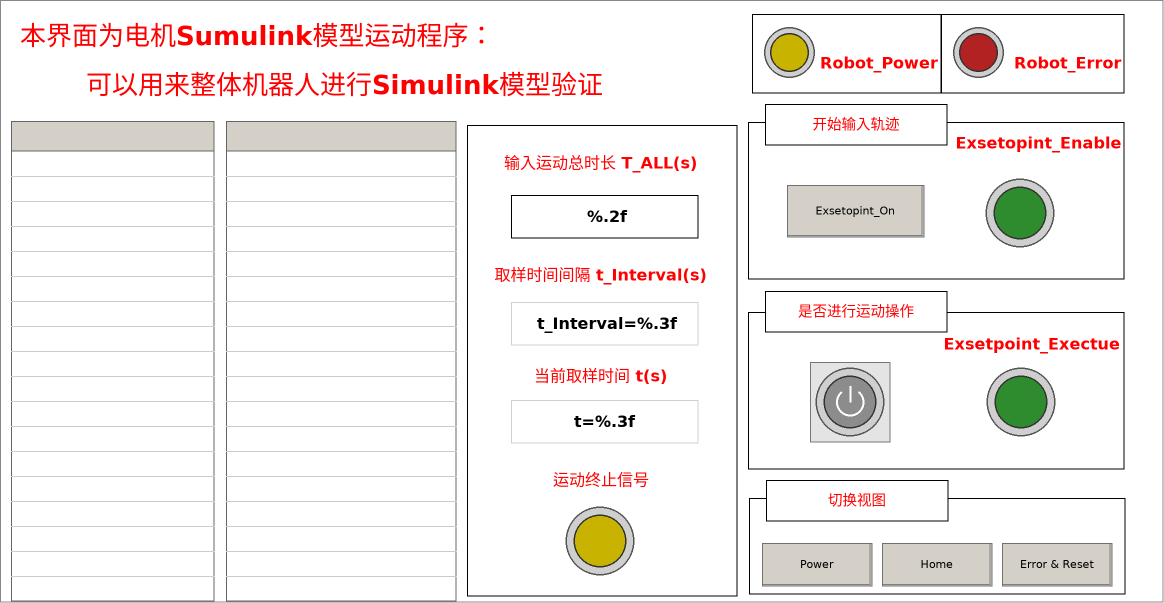
VISUALIZATION Visu_SimulinkMove  // 1164x603
    Rectangle (749,498 376x96)
    Rectangle (766,480 182x41), "切换视图"
    Button (762,543 110x43), "Power"
        OnMouseClick: change screen: Visu_Power
    Button (1002,543 110x43), "Error & Reset"
        OnMouseClick: change screen: Visu_Reset
    Button (882,543 110x43), "Home"
        OnMouseClick: change screen: Visu_Home
    Rectangle (467,125 270x471)
    Rectangle (752,14 189x79)
    Rectangle (748,312 376x157)
    Label (902,328 260x32), "Exsetpoint_Exectue"
    Rectangle (765,291 182x41), "是否进行运动操作"
    Lamp1 (981,362 80x80), variable: ExSetPoint_Execute, style: Lamp-Lamp1-Green
    PowerSwitch (810,362 80x80), variable: ExSetPoint_Execute, behaviour: TOGGLE, style: Switch-PowerSwitch-Gray
    Rectangle (941,14 183x79)
    Lamp1 (948,23 61x59), variable: Hexapod_Robot.Robot_Error, style: Lamp-Lamp1-Red
    Label (991,47 154x32), "Robot_Error"
    Label (17,15 572x42), "本界面为电机Sumulink模型运动程序："
    Label (83,64 874x42), "可以用来整体机器人进行Simulink模型验证"
    Table (11,121 203x480), data array: Hexapod_Robot.Axis_ActPostion
        p3854506369: Hexapod_Robot.Axis_ActPostion[INDEX]
        p2232123230: Axis_ActPostion[Robot]
    Table (226,121 230x480), data array: Hexapod_Robot.Current_Turque_Value
        p3854506369: Hexapod_Robot.Current_Turque_Value[INDEX]
        p2232123230: Current_Turque_Value[Robot]
    Lamp1 (759,23 61x59), variable: Hexapod_Robot.Robot_Power, style: Lamp-Lamp1-Yellow
    Label (802,47 154x32), "Robot_Power"
    Rectangle (748,122 376x157)
    Rectangle (765,104 182x41), "开始输入轨迹"
    Lamp1 (980,173 80x80), variable: MAIN.ExtSetPointEnable, style: Lamp-Lamp1-Green
    Label (935,127 207x32), "Exsetopint_Enable"
    Rectangle (511,195 187x43), "%.2f", text variable: MAIN.T_All
        OnMouseClick: write MAIN.T_All via Default
    Label (471,147 260x32), "输入运动总时长 T_ALL(s)"
    Textfield (511,400 187x43), "t=%.3f", text variable: MAIN.t
    Label (471,360 260x32), "当前取样时间 t(s)"
    Button (787,185 137x52), "Exsetopint_On"
        toggle MAIN.ExtSetPointEnable
    Lamp1 (560,501 80x80), variable: MAIN.ExtSetPointDisable, style: Lamp-Lamp1-Yellow
    Label (471,464 260x32), "运动终止信号"
    Label (471,259 260x32), "取样时间间隔 t_Interval(s)"
    Textfield (511,302 187x43), "t_Interval=%.3f", text variable: MAIN.t_Interval
        OnMouseClick: write MAIN.t_Interval via Default
END_VISUALIZATION

(* stored: Version 1.1.0.1, ProductVersion 3.1.4020.12
   Visu Visu_SimulinkMove: Id {4953c662-5946-414d-97eb-1dec552a9040} *)
